				ELSE
					// Error: Assignment-ID is false 
					mReturnCode := E_ErrorConv.ASSIGNMENT_ID_WRONG;
					// debug message: '11-000-0000-00-0,  AssignmentID mismatch,  telegram = TTA,  expected = 87654321,  current = 12345678'
					DebugMsg:= '';
					DebugMsg:= CONCAT(DebugMsg, F_AddDividerToSisString(SubsystemRegistry.SubsystemName));
					DebugMsg:= CONCAT(DebugMsg, ',  AssignmentID mismatch');
					DebugMsg:= CONCAT(DebugMsg, DebugTextBlocks.TELEGRAM);
					DebugMsg:= CONCAT(DebugMsg, 'TTA');
					DebugMsg:= CONCAT(DebugMsg, DebugTextBlocks.EXPECTED);
					DebugMsg:= CONCAT(DebugMsg, UDINT_TO_STRING(TU_DataTable[mpTTA^.TU_DataIndex].AssignmentID)  );
					DebugMsg:= CONCAT(DebugMsg, DebugTextBlocks.CURRENT);
					DebugMsg:= CONCAT(DebugMsg, UDINT_TO_STRING(mpTTA^.AssignmentID)  );
					fbDebugMsg.M_SendErrorMsg(mMessage := DebugMsg);
				END_IF

			// Checks okay, its allowed to takeover data
			ELSE
				mTU_DataIndex := mpTTA^.TU_DataIndex;
			END_IF
		END_IF
	ELSE
		// Error: No corresponding data set found
		mReturnCode := E_ErrorConv.TU_DATA_INDEX_FREE;
		// debug message: '11-000-0000-00-0,  no corresponding dataset ,  telegram = TTA,  TU_DataIndex = 8'
		DebugMsg:= '';
		DebugMsg:= CONCAT(DebugMsg, F_AddDividerToSisString(SubsystemRegistry.SubsystemName));
		DebugMsg:= CONCAT(DebugMsg, ',  no corresponding dataset');
		DebugMsg:= CONCAT(DebugMsg, DebugTextBlocks.TELEGRAM);
		DebugMsg:= CONCAT(DebugMsg, 'TTA');
		DebugMsg:= CONCAT(DebugMsg, DebugTextBlocks.TU_DATA_INDEX);
		DebugMsg:= CONCAT(DebugMsg, DINT_TO_STRING(mpTTA^.TU_DataIndex)  );
		fbDebugMsg.M_SendErrorMsg(mMessage := DebugMsg);
	
	END_IF
END_IF


(**************************************************************************************
already an error -> cancel processing
***************************************************************************************)
IF mReturnCode <> 0 THEN
	TTC.Position    := mpTTA^.Position;
	TTC.TU_DataIndex:= mTU_DataIndex;
	TTC.MsgSequence := mpTTA^.MsgSequence;
	TTC.TU_ID       := mpTTA^.TU_ID;
	TTC.AssignmentID:= mpTTA^.AssignmentID;
	TTC.ReturnCode  := mReturnCode;
	M_SendData(meChannel:= meChannelSrc, 
	mMsgType := E_ITC_MsgTypeConv.TRANSPORT_TASK_COMPLETE, 
	mpData   := ADR(TTC),
	mLen     := SIZEOF(TTC));
	// debug message already sent
	RETURN;
END_IF


(**************************************************************************************
Check destinations
***************************************************************************************)
// Go through all destinations
FOR Idx := 1 TO mpTTA^.NumberOfDestinations DO			
	mDestinationPosition[Idx] := F_SearchFunctionPosition(Position := mpTTA^.Destination[Idx]);		
	// Check destination is invalid
	IF mDestinationPosition[Idx].eFunctionNumber = E_FunctionNumber.F_BEGIN_FUNCTION THEN
		// Destination invalid
		TTC.Position    := mpTTA^.Position;
		TTC.TU_DataIndex:= mTU_DataIndex;
		TTC.MsgSequence := mpTTA^.MsgSequence;
		TTC.TU_ID       := mpTTA^.TU_ID;
		TTC.AssignmentID:= mpTTA^.AssignmentID;
		TTC.ReturnCode  := E_ErrorConv.DESTINATION_INVALID;
		M_SendData(meChannel:= meChannelSrc, 
		mMsgType := E_ITC_MsgTypeConv.TRANSPORT_TASK_COMPLETE, 
		mpData   := ADR(TTC),
		mLen     := SIZEOF(TTC));
		// debug message: '11-000-0000-00-0,  unknown destination addressed,  telegram = TTA,  destination = 99-999-9999-99-9'
		DebugMsg:= '';
		DebugMsg:= CONCAT(DebugMsg, F_AddDividerToSisString(mpTTA^.Position));
		DebugMsg:= CONCAT(DebugMsg, ',  unknown destination addressed');
		DebugMsg:= CONCAT(DebugMsg, DebugTextBlocks.TELEGRAM);
		DebugMsg:= CONCAT(DebugMsg, 'TTA');
		DebugMsg:= CONCAT(DebugMsg, DebugTextBlocks.DESTINATION);
		DebugMsg:= CONCAT(DebugMsg, F_AddDividerToSisString(mpTTA^.Destination[Idx])  );
		fbDebugMsg.M_SendErrorMsg(mMessage := DebugMsg);
		// debug message just sent
		RETURN;
	END_IF
END_FOR


(**************************************************************************************
Determine TU data index
***************************************************************************************)
(* Adding unknown TU data is only allowed if:
- TU-ID is unknown and no assignment-ID is present
- Assignment-ID is unknown and no TU-ID is present
- Assignment-ID and TU-ID is unknown *)
IF (mpTTA^.TU_ID = Conveyor.TU_ID_UNKNOWN AND NOT mAssignmentID_Present) OR
(mpTTA^.AssignmentID = Conveyor.ASSIGNMENT_ID_UNKNOWN AND NOT mTU_ID_Present) OR
(mpTTA^.TU_ID = TU_ID_UNKNOWN AND mpTTA^.AssignmentID = ASSIGNMENT_ID_UNKNOWN) THEN
	// Unknown requests need to be mandatory sent to a position
	IF NOT mRequestForPosition THEN
		//Error: no position request!
		mReturnCode := E_ErrorConv.TU_ID_WRONG;
		// debug message: '11-000-0000-00-0,  no position request,  telegram = TTA'
		DebugMsg:= '';
		DebugMsg:= CONCAT(DebugMsg, F_AddDividerToSisString(SubsystemRegistry.SubsystemName));
		DebugMsg:= CONCAT(DebugMsg, ',  no position request');
		DebugMsg:= CONCAT(DebugMsg, DebugTextBlocks.TELEGRAM);
		DebugMsg:= CONCAT(DebugMsg, 'TTA');
		fbDebugMsg.M_SendErrorMsg(mMessage := DebugMsg);
	
	// If the corresponding position contains no data
	ELSIF mTU_DataIndexPosition = 0 THEN
		// Try insert TU-Data
		mTU_DataIndex := F_InsertTU_Data(
		eFunctionNumber := Position.eFunctionNumber,
		ZoneNumber 		:= Position.ZoneNumber);

		// No free TU Index was found
		IF mTU_DataIndex = 0 THEN
			// Error: No free TU-DataIndex
			mReturnCode := E_ErrorConv.NO_FREE_TU_DATA_SET;
			// debug message: '11-000-0000-00-0,  no free data index,  telegram = TTA,  TuID = 012345,  AssignmentID = 87654321'
			DebugMsg:= '';
			DebugMsg:= CONCAT(DebugMsg, F_AddDividerToSisString(mpTTA^.Position));
			DebugMsg:= CONCAT(DebugMsg, ',  no free data index');
			DebugMsg:= CONCAT(DebugMsg, DebugTextBlocks.TELEGRAM);
			DebugMsg:= CONCAT(DebugMsg, 'TTA');
			DebugMsg:= CONCAT(DebugMsg, DebugTextBlocks.TUID);
			DebugMsg:= CONCAT(DebugMsg, mpTTA^.TU_ID);
			DebugMsg:= CONCAT(DebugMsg, DebugTextBlocks.ASSIGNMENTID);
			DebugMsg:= CONCAT(DebugMsg, UDINT_TO_STRING(mpTTA^.AssignmentID) );
			fbDebugMsg.M_SendErrorMsg(mMessage := DebugMsg);
		END_IF
	// Otherwise
	ELSE
		// Use existing index
		mTU_DataIndex := mTU_DataIndexPosition;
	END_IF

// Otherwise the telegram contains valid IDs
ELSE
	(* If the received telegram contains two valid
	IDs (Assignment and TU) - both have to be equal to the found index. *)
	IF mTU_DataIndex > 0 AND mAssignmentID_Index > 0 THEN
		IF mTU_DataIndex <> mAssignmentID_Index THEN
			mReturnCode := E_ErrorConv.WRONG_VALUE;	
			// debug message: '11-000-0000-00-0,  AssignmentID mismatch,  telegram = TTA,  expected = 87654321,  current = 12345678'
			DebugMsg:= '';
			DebugMsg:= CONCAT(DebugMsg, F_AddDividerToSisString(mpTTA^.Position));
			DebugMsg:= CONCAT(DebugMsg, ',  AssignmentID mismatch');
			DebugMsg:= CONCAT(DebugMsg, DebugTextBlocks.TELEGRAM);
			DebugMsg:= CONCAT(DebugMsg, 'TTA');
			DebugMsg:= CONCAT(DebugMsg, DebugTextBlocks.EXPECTED);
			DebugMsg:= CONCAT(DebugMsg, UDINT_TO_STRING(TU_DataTable[mTU_DataIndex].AssignmentID)  );
			DebugMsg:= CONCAT(DebugMsg, DebugTextBlocks.CURRENT);
			DebugMsg:= CONCAT(DebugMsg, UDINT_TO_STRING(mpTTA^.AssignmentID)  );
			fbDebugMsg.M_SendErrorMsg(mMessage := DebugMsg);
		END_IF

	// If an index based on the assignment-ID was found
	ELSIF mAssignmentID_Index > 0 THEN
		(*  Check if the TU-ID of the found index is unknown.
		Equal to telegram is not needed, because then an index should be found. *)
		IF TU_DataTable[mAssignmentID_Index].TU_ID.ASCII = Conveyor.TU_ID_UNKNOWN THEN
			// Use assignment index
			mTU_DataIndex := mAssignmentID_Index;
		ELSE
			// TU-ID of the found slot does not match
			mReturnCode := E_ErrorConv.TU_ID_WRONG;	
			// debug message: '11-001-0120-01-0,  TuID mismatch,  telegram = TTA,  expected = 112233,  current = 332211'
			DebugMsg:= '';
			DebugMsg:= CONCAT(DebugMsg, F_AddDividerToSisString(mpTTA^.Position));
			DebugMsg:= CONCAT(DebugMsg, ',  TuID mismatch');
			DebugMsg:= CONCAT(DebugMsg, DebugTextBlocks.TELEGRAM);
			DebugMsg:= CONCAT(DebugMsg, 'TTA');
			DebugMsg:= CONCAT(DebugMsg, DebugTextBlocks.EXPECTED);
			DebugMsg:= CONCAT(DebugMsg, TU_DataTable[mAssignmentID_Index].TU_ID.ASCII);
			DebugMsg:= CONCAT(DebugMsg, DebugTextBlocks.CURRENT);
			DebugMsg:= CONCAT(DebugMsg, mpTTA^.TU_ID);
			fbDebugMsg.M_SendErrorMsg(mMessage := DebugMsg);
		END_IF

	// When an index based on the TU-ID was found
	ELSIF mTU_DataIndex > 0 THEN
		(* Check if the Assignment-ID of the found index is unknown.
		Equal to telegram is not needed, because then an index should be found. *)
		IF TU_DataTable[mTU_DataIndex].AssignmentID = Conveyor.ASSIGNMENT_ID_UNKNOWN THEN
			// Keep index (mTU_DataIndex)
			;
		ELSE
			// TU-ID of the found slot does not match
			mReturnCode := E_ErrorConv.ASSIGNMENT_ID_WRONG;	
			// debug message: '11-000-0000-00-0,  AssignmentID mismatch,  telegram = TTA,  expected = 87654321,  current = 12345678'
			DebugMsg:= '';
			DebugMsg:= CONCAT(DebugMsg, F_AddDividerToSisString(mpTTA^.Position));
			DebugMsg:= CONCAT(DebugMsg, ',  AssignmentID mismatch');
			DebugMsg:= CONCAT(DebugMsg, DebugTextBlocks.TELEGRAM);
			DebugMsg:= CONCAT(DebugMsg, 'TTA');
			DebugMsg:= CONCAT(DebugMsg, DebugTextBlocks.EXPECTED);
			DebugMsg:= CONCAT(DebugMsg, UDINT_TO_STRING(TU_DataTable[mTU_DataIndex].AssignmentID)  );
			DebugMsg:= CONCAT(DebugMsg, DebugTextBlocks.CURRENT);
			DebugMsg:= CONCAT(DebugMsg, UDINT_TO_STRING(mpTTA^.AssignmentID)  );
			fbDebugMsg.M_SendErrorMsg(mMessage := DebugMsg);
		END_IF
	END_IF

	IF mReturnCode = 0 THEN
		// If a data index is found
		IF mTU_DataIndex > 0 THEN
			// If the request is for a position
			IF mRequestForPosition THEN
				// Check if this index belongs already to a position	
				mOtherPosition :=	F_SearchPositionOfTU_Index( 
				TU_DataIndex 			:= mTU_DataIndex,
				eStartFunctionNumber	:= E_FunctionNumber.F_BEGIN_FUNCTION);
				
				// If the index was found on another position
				IF (mOtherPosition.eFunctionNumber > E_FunctionNumber.F_BEGIN_FUNCTION OR	
				mOtherPosition.ZoneNumber > 0) AND 
				mOtherPosition.eFunctionNumber <> Position.eFunctionNumber THEN
					// Error: Index found on another location
					mReturnCode := E_ErrorConv.INDEX_MATCH_WITH_POSITION;
					// debug message: '11-000-0000-00-0,  data index found on another location,  telegram = TTA,  position = 99-999-9999-99-9,  TU_DataIndex = 3,  TuID = 012345,  AssignmentID = 87654321'
					DebugMsg:= '';
					DebugMsg:= CONCAT(DebugMsg, F_AddDividerToSisString(mpTTA^.Position));
					DebugMsg:= CONCAT(DebugMsg, ',  data index found on another location');
					DebugMsg:= CONCAT(DebugMsg, DebugTextBlocks.TELEGRAM);
					DebugMsg:= CONCAT(DebugMsg, 'TTA');
					DebugMsg:= CONCAT(DebugMsg, DebugTextBlocks.POSITION);
					DebugMsg:= CONCAT(DebugMsg, F_AddDividerToSisString(mOtherPosition.PositionName));
					DebugMsg:= CONCAT(DebugMsg, F_CreateTU_DataString(TU_DataIndex:= mTU_DataIndex));
					fbDebugMsg.M_SendErrorMsg(mMessage := DebugMsg);
	
					FCQ.Code:= E_ITC_FunctionControlCode.SET_ERROR;
					FCQ.Variable := INT_TO_DINT(mReturnCode);
					
					// Set corresponding position to error
					M_ProcessToFunction(
					meFunctionNumber	:= Position.eFunctionNumber,
					meChannelSrc		:= meChannelSrc,
					mMsgType			:= E_ITC_MsgTypeConv.FUNCTION_CONTROL_REQUEST,
					mpData				:= ADR(FCQ),
					mLen				:= SIZEOF(FCQ));
					
					M_ProcessToFunction(
					meFunctionNumber	:= mOtherPosition.eFunctionNumber,
					meChannelSrc		:= meChannelSrc,
					mMsgType			:= E_ITC_MsgTypeConv.FUNCTION_CONTROL_REQUEST,
					mpData				:= ADR(FCQ),
					mLen				:= SIZEOF(FCQ));
				END_IF
			END_IF
	
		// If the corresponding position consists of an empty TU-Data set, use that one
		ELSIF mTU_DataIndexPosition > 0 THEN
			mTU_DataIndex := mTU_DataIndexPosition;
		ELSE
			// Try insert TU-Data
			mTU_DataIndex := F_InsertTU_Data(
								eFunctionNumber := Position.eFunctionNumber,
								ZoneNumber 		:= Position.ZoneNumber);
			
			// No free TU Index was found
			IF mTU_DataIndex = 0 THEN
				// Error: No free TU-DataIndex
				mReturnCode := E_ErrorConv.NO_FREE_TU_DATA_SET;
				// debug message: '11-000-0000-00-0,  no free data index,  telegram = TTA,  TuID = 012345,  AssignmentID = 87654321'
				DebugMsg:= '';
				DebugMsg:= CONCAT(DebugMsg, F_AddDividerToSisString(mpTTA^.Position));
				DebugMsg:= CONCAT(DebugMsg, ',  no free data index');
				DebugMsg:= CONCAT(DebugMsg, DebugTextBlocks.TELEGRAM);
				DebugMsg:= CONCAT(DebugMsg, 'TTA');
				DebugMsg:= CONCAT(DebugMsg, DebugTextBlocks.TUID);
				DebugMsg:= CONCAT(DebugMsg, mpTTA^.TU_ID);
				DebugMsg:= CONCAT(DebugMsg, DebugTextBlocks.ASSIGNMENTID);
				DebugMsg:= CONCAT(DebugMsg, UDINT_TO_STRING(mpTTA^.AssignmentID) );
				fbDebugMsg.M_SendErrorMsg(mMessage := DebugMsg);
			END_IF
		END_IF
	END_IF
END_IF


(**************************************************************************************
already an error -> cancel processing
***************************************************************************************)
IF mReturnCode <> 0 THEN
	TTC.Position    := mpTTA^.Position;
	TTC.TU_DataIndex:= mTU_DataIndex;
	TTC.MsgSequence := mpTTA^.MsgSequence;
	TTC.TU_ID       := mpTTA^.TU_ID;
	TTC.AssignmentID:= mpTTA^.AssignmentID;
	TTC.ReturnCode  := mReturnCode;
	M_SendData(meChannel:= meChannelSrc, 
	mMsgType := E_ITC_MsgTypeConv.TRANSPORT_TASK_COMPLETE, 
	mpData   := ADR(TTC),
	mLen     := SIZEOF(TTC));
	// debug message already sent
	RETURN;
END_IF


(**************************************************************************************
If no TU_DataIndex is available
***************************************************************************************)
IF mTU_DataIndex <= 0 THEN
	RETURN;  // debug message already sent
END_IF


(**************************************************************************************
Update TU data -> process TTA
***************************************************************************************)
// Fill in the received TU-Data 
TU_DataTable[mTU_DataIndex].DataSet.DataPresent := TRUE;
TU_DataTable[mTU_DataIndex].DataSet.JobPresent  := FALSE;

IF mTU_ID_Present THEN
	TU_DataTable[mTU_DataIndex].TU_ID.HashCode := F_CreateHashCode(mpTTA^.TU_ID);
	TU_DataTable[mTU_DataIndex].TU_ID.ASCII    := mpTTA^.TU_ID;
ELSE
	TU_DataTable[mTU_DataIndex].TU_ID.HashCode := F_CreateHashCode(Conveyor.TU_ID_UNKNOWN);
	TU_DataTable[mTU_DataIndex].TU_ID.ASCII    := Conveyor.TU_ID_UNKNOWN;
END_IF

IF mAssignmentID_Present THEN
	TU_DataTable[mTU_DataIndex].AssignmentID := mpTTA^.AssignmentID;
ELSE
	TU_DataTable[mTU_DataIndex].AssignmentID := Conveyor.ASSIGNMENT_ID_UNKNOWN;
END_IF

TU_DataTable[mTU_DataIndex].DataSet.Dimension.Height:= mpTTA^.Height;
TU_DataTable[mTU_DataIndex].DataSet.Dimension.Length:= mpTTA^.Length;
TU_DataTable[mTU_DataIndex].DataSet.Dimension.Weight:= mpTTA^.Weight;
TU_DataTable[mTU_DataIndex].DataSet.Dimension.Width := mpTTA^.Width;
TU_DataTable[mTU_DataIndex].DataSet.Orientation		:= mpTTA^.Orientation;
TU_DataTable[mTU_DataIndex].DataSet.TU_Parameter	:= mpTTA^.TU_Parameter;
TU_DataTable[mTU_DataIndex].DataSet.TU_Type 		:= mpTTA^.TU_Type;
TU_DataTable[mTU_DataIndex].DataSet.IO_Data 		:= mpTTA^.IO_Data;
TU_DataTable[mTU_DataIndex].DataSet.LowerLimit 		:= mpTTA^.LowerLimit;
TU_DataTable[mTU_DataIndex].DataSet.UpperLimit 		:= mpTTA^.UpperLimit;
TU_DataTable[mTU_DataIndex].DataSet.Sequence 		:= mpTTA^.Sequence;			
TU_DataTable[mTU_DataIndex].DataSet.SubSequence 	:= mpTTA^.SubSequence;			
TU_DataTable[mTU_DataIndex].DataSet.SequenceSize 	:= mpTTA^.SequenceSize;		
TU_DataTable[mTU_DataIndex].DataSet.GroupID 		:= mpTTA^.GroupID;			
TU_DataTable[mTU_DataIndex].DataSet.GroupSize 		:= mpTTA^.GroupSize;	
TU_DataTable[mTU_DataIndex].DataSet.DestinationSlot := mpTTA^.DestinationSlot;	
TU_DataTable[mTU_DataIndex].DataSet.NumberOfDest	:= mpTTA^.NumberOfDestinations;

// Clear destination table 
MEMSET(destAddr := ADR(TU_DataTable[mTU_DataIndex].Destination), fillByte := 0, n := SIZEOF(TU_DataTable[mTU_DataIndex].Destination));


// debug message: '11-000-0000-00-0,  new destination assigned,  telegram = TTA,  TU_DataIndex = 3,  TuID = 123456,  AssignmentID = 87654321,  destination = 99-999-9999-99-9,  destination = 99-999-9999-99-9'
DebugMsg:= '';
DebugMsg:= CONCAT(DebugMsg, F_AddDividerToSisString(mpTTA^.Position));
DebugMsg:= CONCAT(DebugMsg, ',  new destination assigned');
DebugMsg:= CONCAT(DebugMsg, DebugTextBlocks.TELEGRAM);
DebugMsg:= CONCAT(DebugMsg, 'TTA');
IF NOT mRequestForPosition THEN
	mOtherPosition:= F_SearchPositionOfTU_Index(TU_DataIndex        := mTU_DataIndex,
	eStartFunctionNumber:= F_BEGIN_FUNCTION);
	DebugMsg:= CONCAT(DebugMsg, DebugTextBlocks.POSITION);
	DebugMsg:= CONCAT(DebugMsg, F_AddDividerToSisString(mOtherPosition.PositionName));
END_IF
DebugMsg:= CONCAT(DebugMsg, F_CreateTU_DataString(TU_DataIndex:= mTU_DataIndex));

// Fill in the destinations 
mDestIndex := 1;
FOR Idx := 1 TO mpTTA^.NumberOfDestinations DO
	// Destination was found 
	IF mDestinationPosition[Idx].eFunctionNumber <> E_FunctionNumber.F_BEGIN_FUNCTION THEN
		TU_DataTable[mTU_DataIndex].DataSet.JobPresent := TRUE;
		TU_DataTable[mTU_DataIndex].Destination[mDestIndex].eFunctionNumber := mDestinationPosition[Idx].eFunctionNumber;
		TU_DataTable[mTU_DataIndex].Destination[mDestIndex].ZoneNumber 		:= mDestinationPosition[Idx].ZoneNumber;
		TU_DataTable[mTU_DataIndex].Destination[mDestIndex].PositionName	:= mpTTA^.Destination[Idx];
		// debug message
		DebugMsg:= CONCAT(DebugMsg, DebugTextBlocks.DESTINATION);
		DebugMsg:= CONCAT(DebugMsg, F_AddDividerToSisString(mpTTA^.Destination[Idx]));
		// continue
		mDestIndex := mDestIndex + 1;
	ELSE
		// Check if it's an external destination
		IF mVirtualDestinationPosition[Idx].eFunctionNumber <> E_FunctionNumber.F_BEGIN_VIRTUAL_FUNCTION THEN
			TU_DataTable[mTU_DataIndex].DataSet.JobPresent := TRUE;
			TU_DataTable[mTU_DataIndex].Destination[mDestIndex].eFunctionNumber 	:= mVirtualDestinationPosition[Idx].eFunctionNumber;
			TU_DataTable[mTU_DataIndex].Destination[mDestIndex].ZoneNumber 			:= 0;
			TU_DataTable[mTU_DataIndex].Destination[mDestIndex].PositionName		:= mpTTA^.Destination[Idx];
			// debug message
			DebugMsg:= CONCAT(DebugMsg, DebugTextBlocks.DESTINATION);
			DebugMsg:= CONCAT(DebugMsg, F_AddDividerToSisString(mpTTA^.Destination[Idx]));
			// continue
			mDestIndex := mDestIndex + 1;
		END_IF
	END_IF
END_FOR

// fire debug message only when if destination exists
IF mDestIndex <> 0 THEN
	fbDebugMsg.M_SendInfoMsg(mMessage := DebugMsg);
END_IF


// Update time stamp 
TU_DataTable[mTU_DataIndex].TimeStamp.eInsertFunctionNumber := E_FunctionNumber.F_BEGIN_FUNCTION;
TU_DataTable[mTU_DataIndex].TimeStamp.InsertZoneNumber := 0;
TU_DataTable[mTU_DataIndex].TimeStamp.InsertDateTime       := System.fbSystemTime.TIMESTR;

// If TTA was sent to a Position 
IF mRequestForPosition THEN
	Data.Init := TRUE;
	Data.TU_DataIndex := mTU_DataIndex;
	Data.ZoneNumber := Position.ZoneNumber;
	
	// Forward to position
	M_ProcessToFunction(meFunctionNumber:= Position.eFunctionNumber, 
						meChannelSrc	:= meChannelSrc, 
						mMsgType		:= E_ITC_MsgTypeConv.ADD_TU_DATA,
						mpData			:= ADR(Data), 
						mLen			:= SIZEOF(Data));
	
	// Update TimeStamp position
	TU_DataTable[mTU_DataIndex].TimeStamp.eInsertFunctionNumber := Position.eFunctionNumber;
	TU_DataTable[mTU_DataIndex].TimeStamp.InsertZoneNumber		:= Position.ZoneNumber;
END_IF



(**************************************************************************************
If position number and zone index is identical  (position = destination)
***************************************************************************************)
// if TTA was send to subsystem -> use TUs position
IF NOT mRequestForPosition THEN
	Position:= mOtherPosition;
END_IF

IF F_DeleteDestination( eFunctionNumber := Position.eFunctionNumber, ZoneNumber := Position.ZoneNumber) THEN

	TTC.Position := mpTTA^.Position;
	TTC.TU_DataIndex := mTU_DataIndex;
	TTC.MsgSequence := mpTTA^.MsgSequence;
	TTC.TU_ID := mpTTA^.TU_ID;
	TTC.AssignmentID := mpTTA^.AssignmentID;
	TTC.ReturnCode := E_ErrorConv.NO_ERROR_CODE;
	
	M_SendData(meChannel:= meChannelSrc, 
	mMsgType := E_ITC_MsgTypeConv.TRANSPORT_TASK_COMPLETE, 
	mpData   := ADR(TTC),
	mLen	 := SIZEOF(TTC));
	
	// debug message: '11-000-0000-00-0,  destination and position are equal,  telegram = TTA'
	DebugMsg:= '';
	DebugMsg:= CONCAT(DebugMsg, F_AddDividerToSisString(mpTTA^.Position));
	DebugMsg:= CONCAT(DebugMsg, ',  destination and position are equal');
	DebugMsg:= CONCAT(DebugMsg, DebugTextBlocks.TELEGRAM);
	DebugMsg:= CONCAT(DebugMsg, 'TTA');
	IF NOT mRequestForPosition THEN
		DebugMsg:= CONCAT(DebugMsg, DebugTextBlocks.POSITION);
		DebugMsg:= CONCAT(DebugMsg, F_AddDividerToSisString(Position.PositionName));
	END_IF
	
	fbDebugMsg.M_SendErrorMsg(mMessage := DebugMsg);
END_IF
END_METHOD

METHOD PROTECTED M_ProcessTUQ : BOOL
(**************************************************************************************
 * 	Application		:	BoxControl Framework
 *	Revision		:	$Revision: 474929 $
 *	Revision date	:	$Date: 2021-04-08 12:45:11 +0200 (tor, 08 apr 2021) $
 *	Last changed by	:	$Author: b7gessa $
 *	URL				:	$URL: http://almscdc.swisslog.com/repo/SWPD/Development/BoxControlFramework/20_Release/tags/R1.12.0/01_Software/BCF/BCF/JumpStart/20_Product/10_BCF/11_Conv/11_Com/11_ITC/FB_ITC_Conveyor.TcPOU $
 *
 *	Purpose			:	Process a received Transport Unit Request telegram.
 *
 * ------------------------------------------------------------------------------------
 *	Copyright Swisslog [IP AG], Switzerland. All rights reserved.
 * 
 * ------------------------------------------------------------------------------------
 *	
 * 	Revision History: 
 *
 * 	VERSION			DATE			INITIALS			DESCRIPTION
 *	0.1				01.01.2001		swl					Example
 *
 **************************************************************************************)
 VAR_INPUT
	meChannelSrc		: E_MFCS_Channel; // Source communicaton channel
	mpTUQ				: POINTER TO ST_ITC_TUQ; // Pointer to TTA
	mLen				: UDINT; // Data length
END_VAR

VAR
	mTU_DataIndex		: DINT; // TU_DataIndex from zone
	mErrorCode			: E_ErrorConv; // ErrorCode
	mPositionName		: STRING(Conveyor.POSITION_STRINGLENGTH); // SIS Position name MM-000-0000-000
	mDestination		: ARRAY [1..Conveyor.NUMBER_OF_DESTINATIONS] OF STRING(Conveyor.POSITION_STRINGLENGTH); // Array of 12 Digit SIS Destinations
	mDestinationIndex	: INT; // DestinationIndex
	mName				: STRING; // temp name
END_VAR
// Initialize
M_ProcessTUQ := TRUE;

// Search TU_DataIndex in the TU-DataTable
mTU_DataIndex := F_SearchTU_ByHashCode(TU_ID := mpTUQ^.TU_ID);

// If TU-ID was found
IF mTU_DataIndex <> 0 THEN
	
	// Get Destinations
	FOR mDestinationIndex := 1 TO TU_DataTable[mTU_DataIndex].DataSet.NumberOfDest DO
		mName := F_GetFunctionName( 
					eFunctionNumber := TU_DataTable[mTU_DataIndex].Destination[mDestinationIndex].eFunctionNumber,
					ZoneNumber		:= TU_DataTable[mTU_DataIndex].Destination[mDestinationIndex].ZoneNumber);
												
		mDestination[mDestinationIndex] := F_ReduceToAlphaNumeric(InputString := mName);
	END_FOR
	
	// Get PositionName from TU_Data
	mPositionName := F_GetFunctionName(
						eFunctionNumber := TU_DataTable[mTU_DataIndex].TimeStamp.eInsertFunctionNumber,
						ZoneNumber		:= 0);
	
	TUR.Position := F_ReduceToAlphaNumeric(InputString := mPositionName);
	TUR.TU_DataIndex := mTU_DataIndex;
	TUR.TU_ID := TU_DataTable[mTU_DataIndex].TU_ID.ASCII;
	TUR.TU_Type := TU_DataTable[mTU_DataIndex].DataSet.TU_Type;
	TUR.AssignmentID := TU_DataTable[mTU_DataIndex].AssignmentID;
	TUR.Length := TU_DataTable[mTU_DataIndex].DataSet.Dimension.Length;
	TUR.Width := TU_DataTable[mTU_DataIndex].DataSet.Dimension.Width;
	TUR.Height := TU_DataTable[mTU_DataIndex].DataSet.Dimension.Height;
	TUR.Weight := TU_DataTable[mTU_DataIndex].DataSet.Dimension.Weight;
	TUR.Orientation := TU_DataTable[mTU_DataIndex].DataSet.Orientation;
	TUR.TU_Parameter := TU_DataTable[mTU_DataIndex].DataSet.TU_Parameter;
	TUR.IO_Data := TU_DataTable[mTU_DataIndex].DataSet.IO_Data;
	TUR.LowerLimit := TU_DataTable[mTU_DataIndex].DataSet.LowerLimit;
	TUR.UpperLimit := TU_DataTable[mTU_DataIndex].DataSet.UpperLimit;
	TUR.Sequence :=	TU_DataTable[mTU_DataIndex].DataSet.Sequence;			
	TUR.SubSequence := TU_DataTable[mTU_DataIndex].DataSet.SubSequence;			
	TUR.SequenceSize :=	TU_DataTable[mTU_DataIndex].DataSet.SequenceSize;		
	TUR.GroupID := TU_DataTable[mTU_DataIndex].DataSet.GroupID;			
	TUR.GroupSize := TU_DataTable[mTU_DataIndex].DataSet.GroupSize;	
	TUR.DestinationSlot :=TU_DataTable[mTU_DataIndex].DataSet.DestinationSlot;		
	TUR.ReturnCode := E_ErrorConv.NO_ERROR_CODE;
	TUR.NumberOfDestinations := TU_DataTable[mTU_DataIndex].DataSet.NumberOfDest;
	TUR.Destination := mDestination;
	
	M_SendData(
		meChannel := meChannelSrc, 
		mMsgType  := E_ITC_MsgTypeConv.TRANSPORT_UNIT_REPORT, 
		mpData    := ADR(TUR),
		mLen	  := SIZEOF(TUR));		
				
ELSE
	TUR.Position := '';
	TUR.TU_DataIndex := 0;
	TUR.TU_ID := mpTUQ^.TU_ID;
	TUR.TU_Type := 0;
	TUR.AssignmentID := 0;
	TUR.Length := 0;
	TUR.Width := 0;
	TUR.Height := 0;
	TUR.Weight := 0;
	TUR.Orientation := '   ';
	TUR.TU_Parameter := 0;
	TUR.IO_Data := 0;
	TUR.LowerLimit := 0;
	TUR.UpperLimit := 0;
	TUR.Sequence :=	0;			
	TUR.SubSequence := 0;			
	TUR.SequenceSize :=	0;		
	TUR.GroupID := 0;			
	TUR.GroupSize := 0;	
	TUR.DestinationSlot :=	0;			
	TUR.ReturnCode := E_ErrorConv.TU_ID_WRONG;
	TUR.NumberOfDestinations := 0;
	TUR.Destination := mDestination;
	
	M_SendData(
		meChannel := meChannelSrc, 
		mMsgType  := E_ITC_MsgTypeConv.TRANSPORT_UNIT_REPORT, 
		mpData    := ADR(TUR),
		mLen	  := SIZEOF(TUR));	
END_IF
END_METHOD

METHOD M_ProcessVIQ : BOOL
(**************************************************************************************
 * 	Application		:	BoxControl Framework
 *	Revision		:	$Revision: 474929 $
 *	Revision date	:	$Date: 2021-04-08 12:45:11 +0200 (tor, 08 apr 2021) $
 *	Last changed by	:	$Author: b7gessa $
 *	URL				:	$URL: http://almscdc.swisslog.com/repo/SWPD/Development/BoxControlFramework/20_Release/tags/R1.12.0/01_Software/BCF/BCF/JumpStart/20_Product/10_BCF/11_Conv/11_Com/11_ITC/FB_ITC_Conveyor.TcPOU $
 *
 *	Purpose			:	Process a received Transport Task Assignment telegram.
 *
 * ------------------------------------------------------------------------------------
 *	Copyright Swisslog [IP AG], Switzerland. All rights reserved.
 * 
 * ------------------------------------------------------------------------------------
 *	
 * 	Revision History: 
 *
 * 	VERSION			DATE			INITIALS			DESCRIPTION
 *	0.1				10.03.2016		Kay Röder			Example
 *
 **************************************************************************************)
VAR_INPUT
	meChannelSrc					: E_MFCS_Channel; // Source communication channel
	mpVIQ							: POINTER TO ST_ITC_VIQ; // Pointer to VIQ
	mLen							: UDINT;
END_VAR
VAR
	meFunctionPosition			: ST_PositionIdent; // Position
	meGroupNumber				: E_GroupNumber; // Group
	meElementNumber				: E_ElementNumber;//Element Number
	meSubsystem					: BOOL;	//Subsystem
	mKeyValuePairs				: ARRAY [1..System.NUMBER_OF_KEYVALUE_PAIRS_VIR] OF ST_ITC_VIR_SET;
END_VAR
// Initialize
M_ProcessVIQ := TRUE;

// Get position from message
meFunctionPosition := F_SearchFunctionPosition(Position := mpVIQ^.Position);
meElementNumber    := F_SearchElementPosition(ElementName := mpVIQ^.Position);
meGroupNumber      := F_SearchGroupNumber(GroupName := mpVIQ^.Position);
meSubsystem 	   := F_EqualSisNames(Name1 := SubsystemRegistry.SubSystemName,
                                    Name2 := mpVIQ^.Position);
														
// If a valid function was found with a valid zone
IF 	meFunctionPosition.eFunctionNumber > E_FunctionNumber.F_BEGIN_FUNCTION AND 
	meFunctionPosition.eFunctionNumber < E_FunctionNumber.F_END_FUNCTION AND 
	meFunctionPosition.ZoneNumber >= 0 AND meFunctionPosition.ZoneNumber <= NUMBER_OF_ZONES_PER_FUNCTION THEN
	
	// Forward to function
	M_ProcessVIQ := M_ProcessToFunction(
						meFunctionNumber	:= meFunctionPosition.eFunctionNumber, 
						meChannelSrc		:= meChannelSrc, 
						mMsgType			:= E_ITC_MsgTypeConv.VISUALIZATION_INFORMATION_REQUEST,
						mpData				:= mpVIQ,
						mLen				:= mLen);

// If a valid element was found
ELSIF meElementNumber > E_ElementNumber.E_BEGIN_ELEMENT AND
 	  meElementNumber < E_ElementNumber.E_END_ELEMENT THEN

	// Forward to element
	M_ProcessVIQ := M_ProcessToElement(
						meElementNumber		:= meElementNumber, 
						meChannelSrc		:= meChannelSrc, 
						mMsgType			:= E_ITC_MsgTypeConv.VISUALIZATION_INFORMATION_REQUEST,
						mpData				:= mpVIQ,
						mLen				:= mLen);	

// If a valid group was found
ELSIF meGroupNumber > E_GroupNumber.G_BEGIN_GROUP AND
 	  meGroupNumber < E_GroupNumber.G_END_GROUP THEN

	// Forward to group
	M_ProcessVIQ := M_ProcessToGroup(
						meGroupNumber		:= meGroupNumber, 
						meChannelSrc		:= meChannelSrc, 
						mMsgType			:= E_ITC_MsgTypeConv.VISUALIZATION_INFORMATION_REQUEST,
						mpData				:= mpVIQ,
						mLen				:= mLen);		

// If a valid subsystem was found
ELSIF meSubsystem THEN

	// Forward to subsystem
	M_ProcessVIQ := M_ProcessToSubsystem(
						meChannelSrc		:= meChannelSrc, 
						mMsgType			:= E_ITC_MsgTypeConv.VISUALIZATION_INFORMATION_REQUEST,
						mpData				:= mpVIQ,
						mLen				:= mLen);	
ELSE
	// Unknown Position name received 
	DebugMsg := CONCAT('VIQ: Unknown address', mpVIQ^.Position);
	fbDebugMsg.M_SendErrorMsg(mMessage := DebugMsg); 
	
	// Send VIR - error - no valid Address
	F_ITC_SendVIR(
		eChannelSrc := meChannelSrc,
		Position := mpVIQ^.Position,
		NumOfKeyValuePairs := 1,
		KeyValuePairs	:= mKeyValuePairs);
END_IF
END_METHOD

METHOD M_SendData : BOOL
(**************************************************************************************
 * 	Application		:	BoxControl Framework
 *	Revision		:	$Revision: 474929 $
 *	Revision date	:	$Date: 2021-04-08 12:45:11 +0200 (tor, 08 apr 2021) $
 *	Last changed by	:	$Author: b7gessa $
 *	URL				:	$URL: http://almscdc.swisslog.com/repo/SWPD/Development/BoxControlFramework/20_Release/tags/R1.12.0/01_Software/BCF/BCF/JumpStart/20_Product/10_BCF/11_Conv/11_Com/11_ITC/FB_ITC_Conveyor.TcPOU $
 *
 *	Purpose			:	Send data to MFCS connection
 *
 * ------------------------------------------------------------------------------------
 *	Copyright Swisslog [IP AG], Switzerland. All rights reserved.
 * 
 * ------------------------------------------------------------------------------------
 *	
 * 	Revision History: 
 *
 * 	VERSION			DATE			INITIALS			DESCRIPTION
 *	0.1				01.01.2001		swl					Example
 *
 **************************************************************************************)
VAR_INPUT
	meChannel				: E_MFCS_Channel; // Channel to forward msg
	mMsgType				: INT; // Msg type
	mpData					: PVOID; // Data pointer
	mLen					: UDINT; // Data length
END_VAR

VAR
	mMFCS_Instance			: ITF_MFCS; // Instance to compare valid interfaces
END_VAR
// INitialize
M_SendData := TRUE;

// If communication with single source
IF meChannel <> 0 THEN
	IF __QUERYINTERFACE(fbMFCS_Channel[meChannel], mMFCS_Instance) THEN
		// Forward data to MFCS channel
		M_SendData := fbMFCS_Channel[meChannel].M_SendData(
						meChannelSrc := meChannel,
						mMsgType  	 := mMsgType,
						mpData	  	 := mpData,
						mLen		 := mLen);
	END_IF			
// Sender unknown - forward to all
ELSE
	FOR Idx := E_MFCS_Channel.BEGIN_CHANNEL + 1 TO E_MFCS_Channel.END_CHANNEL - 1 DO
		IF __QUERYINTERFACE(fbMFCS_Channel[Idx], mMFCS_Instance) THEN
			// Forward data to MFCS channel
			fbMFCS_Channel[Idx].M_SendData(
				meChannelSrc := meChannel,
				mMsgType  	 := mMsgType,
				mpData	  	 := mpData,
				mLen		 := mLen);
		END_IF
	END_FOR
END_IF
END_METHOD

END_FUNCTION_BLOCK

(* stored: Version 1.1.0.1, ProductVersion 3.1.4024.4
   POU FB_ITC_Conveyor: Id {aa14b97a-f6e8-4949-951d-771f47a40135}, SpecialFunc None
   Method M_AddData: Id {97bd1698-f7f3-4381-8356-3f2b98f7ad14}
   Method M_AddTUData: Id {9d8c0b6e-b982-4909-adff-7c0b22c14777}
   Method M_CallITC_Service: Id {e7fd0a60-471b-4fc5-8779-ba4f1d24b5a5}
   Method M_Init: Id {94653a35-9a2f-4969-b664-a69711cf2bfd}
   Method M_ProcessDAQ: Id {41fc67ae-df8a-43bf-bfbb-23bc430ab5be}
   Method M_ProcessDIQ: Id {6215de98-8248-4eb8-95e0-a944e002ab76}
   Method M_ProcessECQ: Id {ef6956ef-4355-4a98-81f6-c035ac6c922a}
   Method M_ProcessESQ: Id {785210f8-d148-4ab9-8635-051b06acf8ea}
   Method M_ProcessFCQ: Id {0cc7e34d-4c93-4815-be00-f94ca171ebfc}
   Method M_ProcessFSQ: Id {80a3a39d-7aea-4b89-979c-99601e42aa01}
   Method M_ProcessGCQ: Id {ba2bd1f7-2f0c-4b43-a739-582127921df7}
   Method M_ProcessGDQ: Id {289d95b4-fc94-4a5d-a83f-820e062f7639}
   Method M_ProcessGSQ: Id {e858bc3f-b9a0-44f9-aeed-0493b693c012}
   Method M_ProcessGVQ: Id {e7debde4-84d4-4532-a58d-a00f68ae87d4}
   Method M_ProcessIRQ: Id {6f8ce5a4-bac5-48cd-9967-0eb935cc9b1d}
   Method M_ProcessMCQ: Id {a498f02a-a60d-471b-9f14-4ae2d58c599e}
   Method M_ProcessRAA: Id {03041e0e-267c-428d-8328-65e566cb344f}
   Method M_ProcessRDQ: Id {57b3e6ab-86e2-4924-9861-1e27f2775098}
   Method M_ProcessSCQ: Id {eda05472-2ea0-4c8f-9b1e-2a937573679a}
   Method M_ProcessSDO: Id {f8bdd0d3-7e7c-41a7-b606-6bddca251bd5}
   Method M_ProcessSIQ: Id {e93637b9-5bb0-48a7-a032-c0de0cfcf7c6}
   Method M_ProcessSSQ: Id {445a4ec0-5cd3-4bca-8611-2c4a7cd05af2}
   Method M_ProcessTDQ: Id {281dea17-5f65-40c7-9949-8b57aa9a490a}
   Method M_ProcessToElement: Id {9f447273-352d-42d2-a622-94689f4b3a90}
   Method M_ProcessToFunction: Id {77340ee0-7e65-41fb-9f14-f411dc0915a6}
   Method M_ProcessToGroup: Id {5359cffe-baa7-40c7-8382-5ee2aa8963f6}
   Method M_ProcessToSubsystem: Id {05a45ffd-c557-4480-b2d2-4c67b13ed8a2}
   Method M_ProcessTTA: Id {7b073972-ad1d-47f3-97e9-1abc61047186}
   Method M_ProcessTUQ: Id {ce476011-be5c-489f-84d6-15851cb09fe5}
   Method M_ProcessVIQ: Id {1f97e3b5-ac7a-40ae-acec-636990da4efb}
   Method M_SendData: Id {179d4b0e-fea9-459b-9670-450fe5d500b5} *)
